FUNCTION_BLOCK FB_4PViciValve
VAR_INPUT
    iAddress : INT;
END_VAR
VAR_OUTPUT
END_VAR
VAR

    // Re-Use Vici Driver Code for 12 port Value
    fbViciDriver  : FB_ViciDriver;
    fbViciSerial  : FB_SerialCommWrapper;
    stViciSerial  : ST_SerialComm;
    stViciVlvCtrl : ST_ViciControl;
    stViciVlvStatus : ST_ViciStatus;
    //
    iNewPos: INT;
    iMapped : INT;


    {attribute 'pytmc' := '
        pv: ReqPos
        io: io
    '}
    iVici1ReqPos : INT;

    {attribute 'pytmc' := '
        pv: SampleNames
        io: io
     '}
     stSampleName : ST_4PViciValveSampleNames;

END_VAR

iNewPos := LIMIT(1, iVici1ReqPos, 4);

stViciVlvCtrl.iReqPos := iNewPos;
stViciVlvCtrl.iAddress := iAddress;
stViciVlvCtrl.iPortCount := 4;
fbViciDriver(
    i_xExecute:= TRUE,
    i_tTimeOut:= t#10s,
    i_stControl:= stViciVlvCtrl,
    iq_stSerialRXBuffer:= stViciSerial.RxBuffer,
    iq_stSerialTXBuffer:= stViciSerial.TxBuffer,
    q_stStatus=> stViciVlvStatus);

IF 	fbViciDriver.q_xDone OR
    fbViciDriver.q_xError OR
    fbViciDriver.q_xTimeout THEN
    (* reset function for next time *)
    fbViciDriver(i_xExecute:=FALSE,
        iq_stSerialRXBuffer:= stViciSerial.RxBuffer,
        iq_stSerialTXBuffer:= stViciSerial.TxBuffer);

END_IF

fbViciSerial(stSerialComm := stViciSerial);

END_FUNCTION_BLOCK

(* stored: Version 1.1.0.1, ProductVersion 3.1.4024.12
   POU FB_4PViciValve: Id {867cd0ab-cbb3-428d-92e9-f85cb5a24957}, SpecialFunc None *)
